Yaskawa INFORM job: pipe_junction_cone_program.JBI

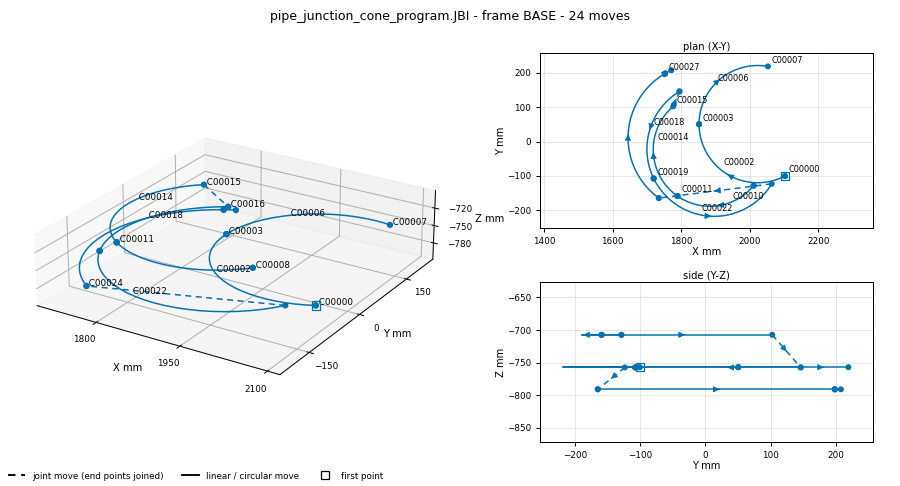
[picture p0: tool path of pipe_junction_cone_program.JBI in frame BASE, 24 of 36 moves have a stored position in this frame; points joined in program order, loops and branches not executed]
/JOB
//NAME pipe_junction_cone_program
//POS
///NPOS 32,0,32,0,0,0
///TOOL 0
///POSTYPE BASE
///RECTAN
///RCONF 0,0,0,0,0,0,0,0,0,0,0,0,0,0,0,0,0,0,0,0,0,0,0,0
C00000=2102.509112,-100.795978,-756.993000,-62.284019,-90.000000,5.000000
C00001=2102.509112,-100.795978,-756.993000,-62.284019,-90.000000,5.000000
C00002=1912.579527,-80.084010,-756.993000,-130.163093,-89.999999,5.000000
C00003=1851.833774,50.301386,-756.993000,-175.000000,-90.000000,5.000000
C00004=1851.833774,50.301386,-756.993000,-175.000000,-90.000000,5.000000
C00005=1851.833774,50.301386,-756.993000,-175.000000,-90.000000,5.000000
C00006=1895.790490,165.170289,-756.993000,137.995311,-89.999999,5.000000
C00007=2052.827974,219.139451,-756.993000,79.937364,-89.999999,5.000000
C00008=2011.142118,-128.764823,-707.393626,-39.505729,-90.000000,5.000000
C00009=2011.142118,-128.764823,-707.393626,-39.505729,-90.000000,5.000000
C00010=1938.470513,-179.556012,-707.393626,-70.593808,-90.000000,5.000000
C00011=1788.881235,-159.219576,-707.393626,-124.889818,-90.000000,5.000000
C00012=1788.881235,-159.219576,-707.393626,-124.889818,-90.000000,5.000000
C00013=1788.881235,-159.219576,-707.393626,-124.889818,-90.000000,5.000000
C00014=1718.916826,-6.895849,-707.393626,174.229773,-89.999999,5.000000
C00015=1776.338940,102.493531,-707.393626,130.377286,-89.999999,5.000000
C00016=1794.692768,146.047402,-757.398626,121.068875,-90.000000,5.000000
C00017=1794.692768,146.047402,-757.398626,121.068875,-90.000000,5.000000
C00018=1708.579936,36.291859,-757.398626,162.696547,-90.000000,5.000000
C00019=1719.378314,-107.768696,-757.398626,-154.123116,-90.000000,5.000000
C00020=1719.378314,-107.768696,-757.398626,-154.123116,-90.000000,5.000000
C00021=1719.378314,-107.768696,-757.398626,-154.123116,-90.000000,5.000000
C00022=1848.403613,-212.539864,-757.398626,-104.031486,-90.000000,5.000000
C00023=2064.064094,-123.526424,-757.398626,-31.111931,-90.000000,5.000000
C00024=1734.281402,-165.039036,-790.936884,-125.932965,-90.000000,5.000000
C00025=1734.281402,-165.039036,-790.936884,-125.932965,-90.000000,5.000000
C00026=1741.749760,191.567097,-790.936884,123.533439,-90.000000,5.000000
C00027=1752.596294,198.304705,-790.936884,120.161688,-90.000000,5.000000
C00028=1752.596294,198.304705,-790.936884,120.161688,-90.000000,5.000000
C00029=1752.596294,198.304705,-790.936884,120.161688,-90.000000,5.000000
C00030=1767.980826,206.437951,-790.936884,115.565894,-90.000000,5.000000
C00031=1770.764987,207.745694,-790.936884,180.000000,-60.000000,-65.246247
///POSTYPE PULSE
///PULSE
EX00000=324608.0
///POSTYPE PULSE
///PULSE
EC00000=106496.0
EC00001=106496.0
EC00002=106496.0
EC00003=106496.0
EC00004=106496.0
EC00005=106496.0
EC00006=106496.0
EC00007=106496.0
EC00008=324608.0
EC00009=324608.0
EC00010=324608.0
EC00011=324608.0
EC00012=324608.0
EC00013=324608.0
EC00014=324608.0
EC00015=324608.0
EC00016=324608.0
EC00017=324608.0
EC00018=324608.0
EC00019=324608.0
EC00020=324608.0
EC00021=324608.0
EC00022=324608.0
EC00023=324608.0
EC00024=324608.0
EC00025=324608.0
EC00026=324608.0
EC00027=324608.0
EC00028=324608.0
EC00029=324608.0
EC00030=324608.0
EC00031=324608.0
//INST
///DATE 2023/08/15 17:09
///ATTR SC,RW,RJ
////FRAME BASE
///GROUP1 RB1,ST1
NOP
MOVJ P009 EX000 VJ=15.00
MOVJ C00000 EC00000 VJ=15.0
CALL JOB:SPYON
MOVC C00001 EC00001 V=150.0
MOVC C00002 EC00002 V=150.0
MOVC C00003 EC00003 V=150.0
MOVJ C00004 EC00004 VJ=15.0
MOVC C00005 EC00005 V=150.0
MOVC C00006 EC00006 V=150.0
MOVC C00007 EC00007 V=150.0
CALL JOB:SPYOF
MOVJ P009 VJ=15.00
MOVJ C00008 EC00008 VJ=15.0
CALL JOB:SPYON
MOVC C00009 EC00009 V=150.0
MOVC C00010 EC00010 V=150.0
MOVC C00011 EC00011 V=150.0
MOVJ C00012 EC00012 VJ=15.0
MOVC C00013 EC00013 V=150.0
MOVC C00014 EC00014 V=150.0
MOVC C00015 EC00015 V=150.0
MOVJ C00016 EC00016 VJ=15.0
MOVC C00017 EC00017 V=150.0
MOVC C00018 EC00018 V=150.0
MOVC C00019 EC00019 V=150.0
MOVJ C00020 EC00020 VJ=15.0
MOVC C00021 EC00021 V=150.0
MOVC C00022 EC00022 V=150.0
MOVC C00023 EC00023 V=150.0
MOVJ C00024 EC00024 VJ=15.0
MOVC C00025 EC00025 V=150.0
MOVC C00026 EC00026 V=150.0
MOVC C00027 EC00027 V=150.0
MOVJ C00028 EC00028 VJ=15.0
MOVC C00029 EC00029 V=150.0
MOVC C00030 EC00030 V=150.0
MOVC C00031 EC00031 V=150.0
CALL JOB:SPYOF
MOVJ P009 VJ=15.00
MOVL P009 EX00000 V=150.0
END
